SUBAPPLICATION Uebung_075a_AUI (* FPTO Speed + SpeedSet auf UT ausgeben mit AR_Timeout_Zero (Adapter Version) *)
  (* Standard: 61499-2; Description: Copyright (c) 2026 Meisterschulen am Ostbahnhof This program and the accompanying materials are made available under the terms of the Eclipse Public License 2.0 which is available at https://www.eclipse.org/legal/epl-2.0/ SPDX-License-Identifier: EPL-2.0 *)
  (* Version 1.0, 2026-09-17, Franz Höpfinger, Meisterschulen am Ostbahnhof, FPTO (Front PTO) Speed + SpeedSet mit PHYS Skalierung (0.125) und 2x AR_Timeout_Zero Fendt-Schaltung (Adapter Version, analog Krauternter TECU_FPTO.SUB) *)
  PACKAGE Uebungen;
  IMPORT Uebungen::const::UT::TECU::DefaultPool_TECU_Numeric::NumberVariable_TECU_FPTO_Speed_N;
  IMPORT Uebungen::const::UT::TECU::DefaultPool_TECU_Numeric::NumberVariable_TECU_FPTO_SpeedSet_N;
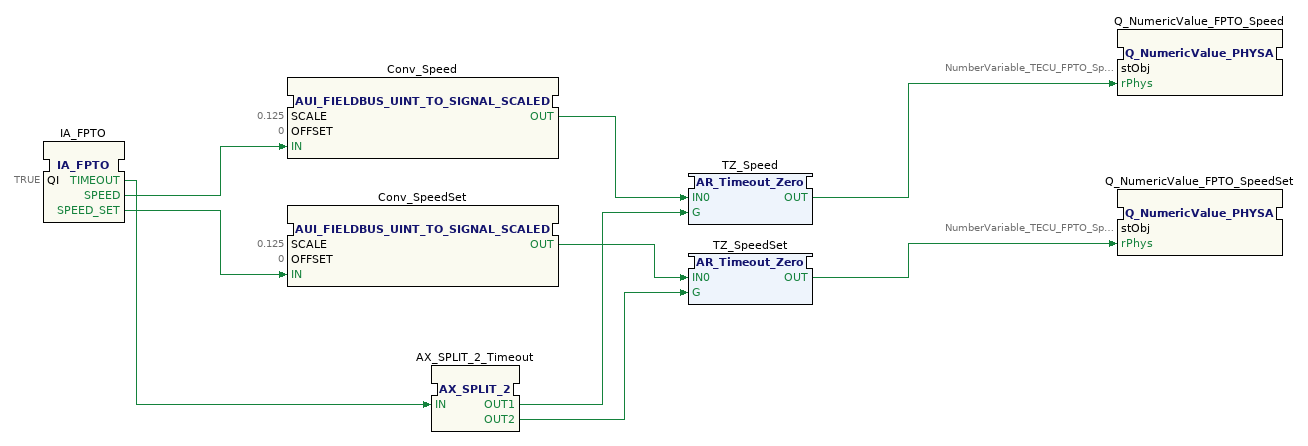
  FBS
    IA_FPTO : isobus::tecu::IA_FPTO(QI := TRUE);
    Conv_Speed : logiBUS::signalprocessing::fieldbus::AUI_FIELDBUS_UINT_TO_SIGNAL_SCALED(SCALE := 0.125, OFFSET := 0);
    Q_NumericValue_FPTO_Speed : isobus::UT::Q::Q_NumericValue_PHYSA(stObj := NumberVariable_TECU_FPTO_Speed_N);
    Conv_SpeedSet : logiBUS::signalprocessing::fieldbus::AUI_FIELDBUS_UINT_TO_SIGNAL_SCALED(SCALE := 0.125, OFFSET := 0);
    Q_NumericValue_FPTO_SpeedSet : isobus::UT::Q::Q_NumericValue_PHYSA(stObj := NumberVariable_TECU_FPTO_SpeedSet_N);
    AX_SPLIT_2_Timeout : adapter::events::unidirectional::AX_SPLIT_2;
  END_FBS
  SUBAPPS
    TZ_Speed : MyLib::sys::AR_Timeout_Zero;
    TZ_SpeedSet : MyLib::sys::AR_Timeout_Zero;
  END_SUBAPPS
  ADAPTER_CONNECTIONS
    IA_FPTO.TIMEOUT TO AX_SPLIT_2_Timeout.IN;
    IA_FPTO.SPEED TO Conv_Speed.IN;
    Conv_Speed.OUT TO TZ_Speed.IN0;
    AX_SPLIT_2_Timeout.OUT1 TO TZ_Speed.G;
    TZ_Speed.OUT TO Q_NumericValue_FPTO_Speed.rPhys;
    IA_FPTO.SPEED_SET TO Conv_SpeedSet.IN;
    Conv_SpeedSet.OUT TO TZ_SpeedSet.IN0;
    AX_SPLIT_2_Timeout.OUT2 TO TZ_SpeedSet.G;
    TZ_SpeedSet.OUT TO Q_NumericValue_FPTO_SpeedSet.rPhys;
  END_CONNECTIONS
END_SUBAPPLICATION
